// Mitsubishi GX Developer project: Traffic Signal Control   PLC: FX1S

PROGRAM MAIN
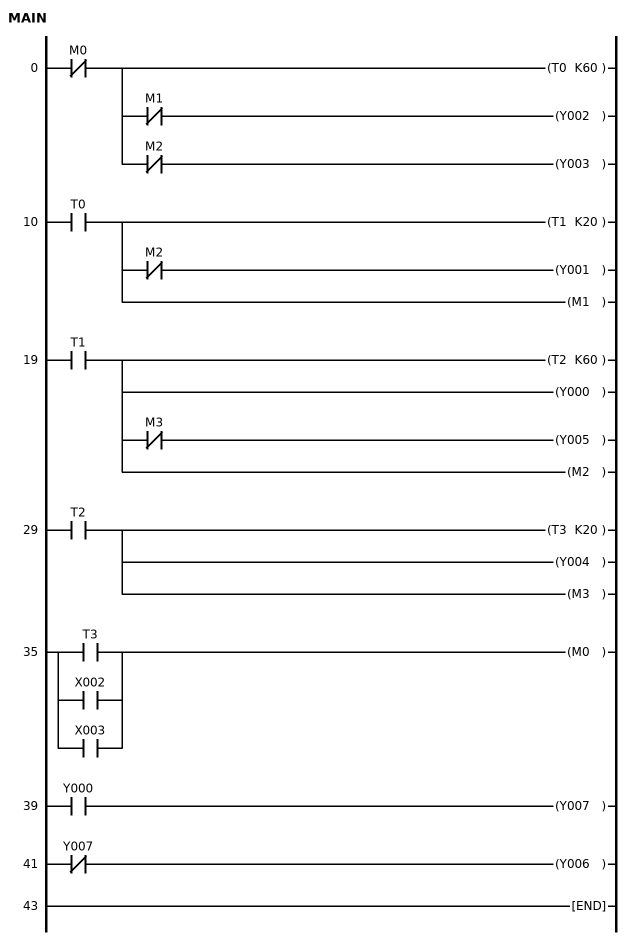
0     LDI     M0
      OUT     T0 K60
      MPS
      ANI     M1
      OUT     Y002
      MPP
      ANI     M2
      OUT     Y003
10    LD      T0
      OUT     T1 K20
      MPS
      ANI     M2
      OUT     Y001
      MPP
      OUT     M1
19    LD      T1
      OUT     T2 K60
      OUT     Y000
      MPS
      ANI     M3
      OUT     Y005
      MPP
      OUT     M2
29    LD      T2
      OUT     T3 K20
      OUT     Y004
      OUT     M3
35    LD      T3
      OR      X002
      OR      X003
      OUT     M0
39    LD      Y000
      OUT     Y007
41    LDI     Y007
      OUT     Y006
43    END
END_PROGRAM
